INTERFACE I_MotionDrive

PROPERTY EnableMode : E_StageEnableMode
GET
END_GET
SET
END_SET
END_PROPERTY

PROPERTY Name : STRING
GET
END_GET
SET
END_SET
END_PROPERTY

END_INTERFACE

(* stored: Version 1.1.0.1
   Itf I_MotionDrive: Id {4f84f724-7938-4847-ac53-18866323f75e}
   Property EnableMode: Id {a11604e5-8855-4fe5-9483-d83f51949d40}
   Get Get: Id {fe8256e3-91a5-4246-b854-e9e12e84b160}
   Set Set: Id {551c9629-a8d7-49a2-9f37-8de0947409ad}
   Property Name: Id {808bc845-b6e4-4963-ab8f-244d15a3cc40}
   Get Get: Id {eef700d5-67cb-4093-abd3-49b2850feb0c}
   Set Set: Id {a8ad97b6-7dbe-4ad8-a2ac-9e24c41ccebb} *)
